{attribute 'qualified_only'}
{attribute 'strict'}
TYPE SafetyDoorStatus:
(
        UNKNOWN := 0, 
		UNLOCKED := 1, 
		LOCKED := 2
);
END_TYPE

(* stored: Version 1.1.0.1, ProductVersion 3.1.4024.12
   DUT SafetyDoorStatus: Id {5a7cc3b2-79bd-4db0-ad2b-bf761093f74a} *)
